FUNCTION_BLOCK FB_ModbusRTU
// Send Modbus Read Request for the first element of the buffer . Then remove the first line when executed ( busy)  and move all the other line to the left. Position 2 becomes position 1 , ...
VAR CONSTANT
	NbElementsBuffer				: UINT := 20;
	
END_VAR

VAR
	Buffer 							: ARRAY[1..NbElementsBuffer] OF Struct_InputRTU ; // Buffer to store actions
	Priority 						: ARRAY[1..NbElementsBuffer] OF UINT; // Array to store priorities
	InitialStruct 					: Struct_InputRTU;
	bInit 							: BOOL;
	ReadRTU1						: FB_ReadModbusRTU_V2;

	KK : UINT;
	
	pBoolNull						: BOOL;
	pIntNull						: INT;
	pArrayNull						: BYTE;

	R_TRIG_Error					: R_TRIG ;
	
END_VAR

IF NOT bInit THEN
	// Empty all structures . 
	M_Init();
ELSE
	
		// ATTENTION , IL NE FAUT PAS ENVOYER UN NOUVEAU MODBUS TANT QUE LE PRECEDENT N EST PAS FINI DE TRAITER .DE MEME IL NE FAUT PAS QUE LE CYCLE D AJOUT DU FIFO SOIT PLUS RAPIDE QUE LE TRAITEMENT DU RTU 
		// TEmpo de 30 s apres une alarmes avant de refaire un essai . il ne faudrait pas que ca bloque les autres commandes .  

		IF priority[1] <> 0 THEN

			ReadRTU1(
				InClockRead := TRUE,
				InStartAddr := Buffer[1].InStartAddr,
				InQuantity := Buffer[1].InQuantity,
				InUnitID := Buffer[1].InUnitID,
				InTimeout := T#500MS,
				InAddrDest := Buffer[1].InBuffer,
				InFunctionRead := Buffer[1].InFunction
			);
		END_IF
		
		
		
		MEMCPY(destAddr := Buffer[1].OutBusy, srcAddr := ADR(ReadRTU1.OutBusy), n := SIZEOF(ReadRTU1.OutBusy));		

		//R_TRIG_Error(CLK:= ReadRTU1.OutErrorMbRead) ; 
		
		IF ReadRTU1.OutbCompleted OR ReadRTU1.OutErrorMbRead THEN	// La lecture s 'est terminée par une erreur ou correcteemnt, on passe à l'element du buffer suivant . 
			MEMCPY(destAddr := Buffer[1].OutError, srcAddr := ADR(ReadRTU1.OutErrorMbRead), n := SIZEOF(ReadRTU1.OutErrorMbRead)); // Copy the errOR  
			MEMCPY(destAddr := Buffer[1].OutErrorId, srcAddr := ADR(ReadRTU1.OutErrorId), n := SIZEOF(ReadRTU1.OutErrorId));
			MEMCPY(destAddr := Buffer[1].OutCompleted, srcAddr := ADR(ReadRTU1.OutbCompleted), n := SIZEOF(ReadRTU1.OutbCompleted));	
			ReadRTU1.InClockRead := FALSE ; 
			ReadRTU1.Reset		:= TRUE ; 
			M_DeleteAction(InLigne := 1);
			//R_TRIG_Error(CLK:= FALSE ) ; 
			
		END_IF
END_IF

METHOD M_AddAction_FIFO : UINT //Method to add an element with a priority using FIFO strategy

VAR_INPUT
	InStruct 		: Struct_InputRTU;		// Structure input
	InPriority 		: UINT;					// Strategy input
END_VAR
VAR_OUTPUT
	OutBusy 		: BOOL;					// Output state of the Method
	OutError 		: BOOL;					// Output error of the Method
	OutErrorID 		: UINT;					//1: Empty input 2: Full Buffer
	OutCompleted 	: BOOL;					// Output state of the Method : not busy and no error
END_VAR
VAR
	KK 				: UINT;
	LineToDelete	: UINT;
END_VAR
OutError 	:= FALSE;
OutBusy 	:= TRUE;

IF NOT (CheckStruct(InStruct1 := InitialStruct, InStruct2 := InStruct)) AND InPriority <> 0 THEN 			// Check that we don't input an empty value
	IF CheckStruct(InStruct1 := buffer[NbElementsBuffer], InStruct2 := InitialStruct) THEN 			// Check that the buffer isn't already full
		FOR KK := 1 TO NbElementsBuffer - 1 DO
			IF NOT CheckStruct(InStruct1 := buffer[NbElementsBuffer-KK], InStruct2 := InitialStruct) AND Priority[NbElementsBuffer-KK] > InPriority THEN 			// If the next position isn't empty  
				buffer[NbElementsBuffer-KK+1] := buffer[NbElementsBuffer-KK]; 		// I replace this position by the next  ( CE PREMIER IF N EST PAS EXECUTER SI TOUTES LES PRIORITES SONT IDENTIQUES . )
				Priority[NbElementsBuffer -KK +1 ] := Priority[NbElementsBuffer-KK];
			ELSE
				IF NOT CheckStruct(InStruct1 := buffer[NbElementsBuffer-KK], InStruct2 := InitialStruct) THEN		// Detect for buffer element that is not empty and assign new element to read to it. 
					buffer[NbElementsBuffer-KK+1] 	:= InStruct;
					M_AddAction_FIFO 				:= NbElementsBuffer-KK+1;
					Priority[NbElementsBuffer-KK+1] := InPriority;
					OutCompleted 		:= TRUE;
					EXIT ;
				END_IF
			END_IF
		END_FOR
		IF NOT Outcompleted THEN
			buffer[1] := InStruct;
			Priority[1] := InPriority;
			OutCompleted := TRUE;
			M_AddAction_Fifo := 1;
		END_IF
	ELSE
		OutErrorID 	:= 2;
		OutError 	:= TRUE;
	END_IF
ELSE
	OutErrorID 	:= 1;
	OutError 	:= TRUE;
END_IF
IF M_VerifActions(OutLigne=>LineToDelete) THEN	// Verifie si il  n ya pas deux fois la meme ligne , sinon, supprime les lignes en doubles . En pratique, forcement la derniere ligne . 
	M_DeleteAction(InLigne := LineToDelete);
END_IF
OutBusy := FALSE;
END_METHOD

METHOD M_DeleteAction : BOOL
VAR_INPUT
	InLigne 	: UINT;			// Input Ligne to delete
END_VAR
VAR_OUTPUT
	OutBusy 		: BOOL;					// Output state of the Method
	OutError 		: BOOL;					// Output error of the Method
	OutErrorID 		: UINT;					// 1: InLigne greater than Buffer size, 2: The buffer ligne is already empty, 3: The buffer is full
	OutCompleted 	: BOOL;					// Output state of the Method : not busy and no error
	
END_VAR

VAR
	KK 				: UINT;
END_VAR
IF InLigne <= NbElementsBuffer THEN // Check the InLigne is in the range of the buffer
	IF NOT checkstruct(InStruct1 := buffer[InLigne], InStruct2 := InitialStruct) THEN	// Check that the buffer ligne is not already empty
		IF checkstruct(InStruct1 := buffer[NbElementsBuffer], InStruct2 := InitialStruct)THEN //check that the buffer is not full
			FOR KK := InLigne TO NbElementsBuffer -1 DO
				Buffer[KK] := buffer[KK + 1] ;
				Priority[KK] := Priority[KK + 1] ;
			END_FOR
		ELSE
			OutError := TRUE;
			OutBusy := FALSE;
			OutCompleted := FALSE;
			OutErrorID := 3;
		END_IF
	ELSE
		OutError := TRUE;
		OutCompleted := FALSE;
		OutBusy := TRUE;
		OutErrorID := 2;
		
	END_IF
ELSE
	OutCompleted := FALSE;
	OutError := TRUE;
	OutBusy := FALSE;
	OutErrorID := 1;
END_IF
END_METHOD

METHOD M_Init : BOOL
VAR
	InStruct : Struct_InputRTU;
END_VAR

// Initialize the structure with empty elements. 

InitialStruct.InBuffer := ADR(pArrayNull);
InitialStruct.OutBusy := ADR(pBoolNull);
InitialStruct.OutCompleted := ADR(pBoolNull);
InitialStruct.OutError := ADR(pBoolNull);
InitialStruct.OutErrorId := ADR(pIntNull);
FOR KK := 1 TO NbElementsBuffer DO 
	Buffer[KK] := InitialStruct;
END_FOR	

bInit := TRUE;
END_METHOD

METHOD M_VerifActions : BOOL // Verifies there is not repeat in the liste : TRUE = At least 2 elements are the same
VAR_OUTPUT
	OutLigne 	 : UINT;
END_VAR

VAR
	KK: UINT;
	JJ: UINT;
	CheckStructValue : BOOL;
END_VAR
FOR KK := 1 TO NbElementsBuffer DO
	FOR JJ := 1 + KK TO NbElementsBuffer DO
		IF CheckStruct(InStruct1 := InitialStruct, instruct2 := buffer[KK]) THEN
			EXIT;
		ELSE
			CheckStructValue :=  checkstruct(InStruct1 := buffer[JJ], InStruct2 := buffer[KK]);
			M_VerifActions := M_VerifActions OR (CheckStructValue ) ;
			OutLigne := SEL(CheckStructValue AND Priority[KK]> priority[JJ], KK, JJ);
		END_IF
	END_FOR
END_FOR
END_METHOD

END_FUNCTION_BLOCK

(* stored: Version 1.1.0.1, ProductVersion 3.1.4024.6
   POU FB_ModbusRTU: Id {0fdf8f63-1c42-4cb9-add2-71a8a8a1b9ac}, SpecialFunc None
   Method M_AddAction_FIFO: Id {3a64f83e-683f-4608-a822-9b1d3979650f}
   Method M_DeleteAction: Id {5cc42d9c-c214-41c2-a7b4-8a98ac5346c8}
   Method M_Init: Id {02a2d7ca-c70e-4236-ad10-a2c8a0852d1d}
   Method M_VerifActions: Id {09ecf2ea-53c8-4c78-8b42-6e6d91e7dbef} *)
